(* PLC project requests_management, Dassault Systèmes ControlBuild 2024x *)
(* stored: creationDateTime 2023-10-03T11:13:40-01:00 *)

FUNCTION_BLOCK bottling_line.requests_management
  VAR_INPUT
    preparationValve1 : BOOL := false;
    preparationValve2 : BOOL := false;
    preparationValve3 : BOOL := false;
    preparationValve4 : BOOL := false;
    preparationPump1 : BOOL := false;
    preparationPump2 : BOOL := false;
    preparationAgitator : BOOL := false;
  END_VAR
  VAR_INPUT
    productionPump1 : BOOL := false;
    productionPump2 : BOOL := false;
    productionValve1 : BOOL := false;
    productionValve2 : BOOL := false;
    productionValve3 : BOOL := false;
    productionValve4 : BOOL := false;
    productionLSAgitator : BOOL := false;
    productionHSAgitator : BOOL := false;
  END_VAR
  VAR_OUTPUT
    pump1 : BOOL := false;
    pump2 : BOOL := false;
    valve1 : BOOL := false;
    valve2 : BOOL := false;
    valve3 : BOOL := false;
    valve4 : BOOL := false;
    loSpeedAgit : BOOL := false;
    hiSpeedAgit : BOOL := false;
  END_VAR

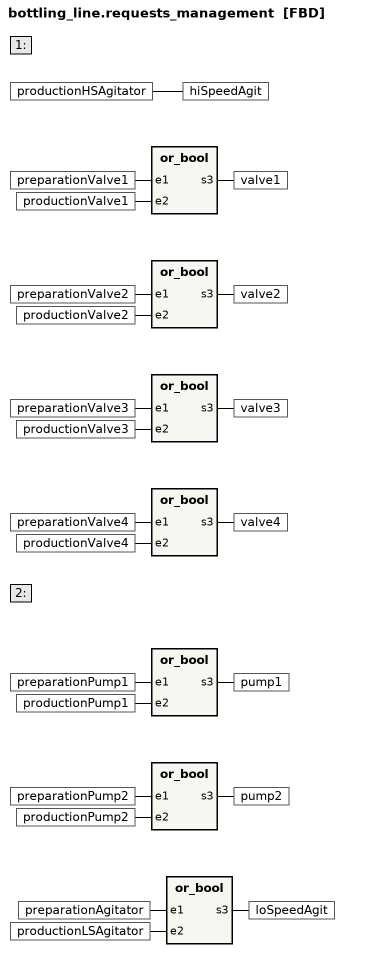
(* FBD diagram, written out as Structured Text *)
1:
2:
valve1 := or_bool(preparationValve1, productionValve1);
pump1 := or_bool(preparationPump1, productionPump1);
valve2 := or_bool(preparationValve2, productionValve2);
pump2 := or_bool(preparationPump2, productionPump2);
valve3 := or_bool(preparationValve3, productionValve3);
loSpeedAgit := or_bool(preparationAgitator, productionLSAgitator);
valve4 := or_bool(preparationValve4, productionValve4);
hiSpeedAgit := productionHSAgitator;
END_FUNCTION_BLOCK
